FUNCTION_BLOCK FB_LamparaAsignada_SFC_2
// La lampara se enciende mientras se acciona el pulsador
VAR
    Lampara AT %Q*: BOOL;
    Pulsador AT %I*: BOOL;
END_VAR

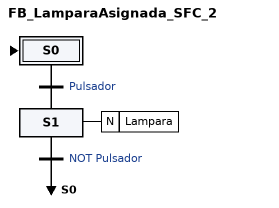
INITIAL_STEP S0:
END_STEP
TRANSITION FROM S0 TO S1
    := Pulsador;
END_TRANSITION
STEP S1:
    Lampara(N);
END_STEP
TRANSITION FROM S1 TO S0
    := NOT Pulsador;
END_TRANSITION

END_FUNCTION_BLOCK

(* stored: Version 1.1.0.1, ProductVersion 3.1.4024.15
   POU FB_LamparaAsignada_SFC_2: Id {bb4f7988-95ce-42ce-b8e0-58fe48877932}, SpecialFunc None *)
